// TIA Portal V20 export
TYPE "typeEnCounter"
TITLE = Energy counter
// Struktur Energy Counter / Structure energy counter
// stored: Access Published
   STRUCT
      activeRate1Imp : LReal;   // Wirkleitungsrate1 Import / Effective rate1 import
      activeRate1Exp : LReal;   // Wirkleitungsrate1 Export / Effective rate1 export
      activeRate2Imp : LReal;   // Wirkleitungsrate2 Import / Effective rate2 import
      activeRate2Exp : LReal;   // Wirkleitungsrate2 Export / Effective rate2 export
      reactiveRate1Imp : LReal;   // Blindleitungsrate1 Import / Reactive rate1 import
      reactiveRate1Exp : LReal;   // Blindleitungsrate1 Export / Reactive rate1 export
      reactiveRate2Imp : LReal;   // Blindleitungsrate2 Import / Reactive rate2 import
      reactiveRate2Exp : LReal;   // Blindleitungsrate2 Export / Reactive rate2 export
      apparentRate1Imp : LReal;   // Scheinleitungsrate1 Import / Apparent rate1import
      apparentRate2Imp : LReal;   // Scheinleitungsrate2 Import / Apparent rate2 import
   END_STRUCT;
END_TYPE
